{attribute 'no_explicit_call' := 'LightOnCommand is a CLASS and must be accessed using methods or properties'}
FUNCTION_BLOCK OnCommand IMPLEMENTS I_Command
VAR
	_onCommand					: I_OnCommand;
END_VAR


// The body of a class must not be used for code.  
// Cyclic code should be called from a method if needed.

METHOD Execute
_onCommand.On();
END_METHOD

METHOD FB_init : BOOL
VAR_INPUT
	bInitRetains : BOOL; // if TRUE, the retain variables are initialized (warm start / cold start)
	bInCopyCode : BOOL;  // if TRUE, the instance afterwards gets moved into the copy code (online change)
	OnCommand			: I_OnCommand;
END_VAR
_onCommand  := OnCommand;
END_METHOD

END_FUNCTION_BLOCK

(* stored: Version 1.1.0.1, ProductVersion 3.1.4024.11
   POU OnCommand: Id {1bf958bb-8da5-4fe5-b211-cd925c9324ef}, SpecialFunc None
   Method Execute: Id {5599378b-6469-4527-9f92-5b5e4c526886}
   Method FB_init: Id {252dd9d1-9b47-4982-9556-4413dd5fe75a} *)
